// TIA Portal project "S7-1500 ile Giyotin Makası Kontrolü Uygulaması" (V18)

(* hardware
DEVICE "S7-1500/ET200MP station_1"  S7-1500 station
   slot 0: "Rail_0"  Rack  6ES7 590-1***0-0AA0
   slot 1: "PLC_1"  CPU 1512C-1 PN  6ES7 512-1CK01-0AB0  V2.8
      slot 3: "CPU display_1"  6ES7591-1AA00-0AA0
      slot 32768: "PROFINET interface_1"  X1
         slot 32769: "Port_1"  X1 P1
         slot 32770: "Port_2"  X1 P2
      slot 34817: "Virtual CP interface port_1"  Virtual CP interface port  Virtual CP interface port
DEVICE "HMI_1"  KTP700 Basic PN
   slot 0: "HMI_1"  KTP700 Basic PN  6AV2 123-2GB03-0AX0  14.0.1.0
   slot 1: "HMI_RT_1"  KTP700 Basic PN  6AV2 123-2GB03-0AX0  14.0.1.0
   slot 5: "HMI_1.IE_CP_1"  PROFINET Interface  14.0.1.0
      slot 1: "PROFINET Interface_1"  PROFINET Interface
         slot 1: "Port_1"  Port
*)

// ===== PLC "PLC_1"  CPU 1512C-1 PN =====

VAR_GLOBAL   // PLC tag table "Default tag table"
   "Stop" AT %M0.0 : Bool;
   "İleri" AT %Q0.0 : Bool;
   "Sınır Anahtarı" AT %M0.1 : Bool;
   "Start_1" AT %M0.2 : Bool;
   "Geri" AT %Q0.1 : Bool;
   "Start_2" AT %M0.3 : Bool;
END_VAR

ORGANIZATION_BLOCK "Main"   // OB1, LAD, ProgramCycle
TITLE = "Main Program Sweep (Cycle)"
{ S7_Optimized_Access := 'TRUE' }
VERSION : 0.1
   VAR_INPUT
      Initial_Call : Bool;   // Initial call of this OB
      Remanence : Bool;   // =True, if remanent data are available
   END_VAR
BEGIN

REGION Network 1: Giyotin makasın ileri-geri yön kontrolü yapılacaktır.
   // 2 starta basınca sistem giyorin sistemi çalışacaktır.
   // Stop+Sınır anahtarı aktif olunca sistem geri gidecek.
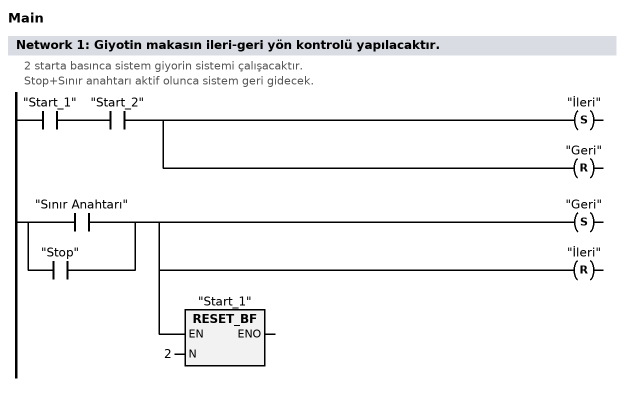
   // no SCL statement known for RBitfield: written as a call
   IF "Start_1" AND "Start_2" THEN
       "İleri" := TRUE;
       "Geri" := FALSE;
   END_IF;
   IF "Sınır Anahtarı" OR "Stop" THEN
       "Geri" := TRUE;
       "İleri" := FALSE;
       RESET_BF(operand := "Start_1", n := 2);
   END_IF;
END_REGION
END_ORGANIZATION_BLOCK

(* ===== HMI "HMI_RT_1" =====
system functions are stored by id; their names below are inferred from use
connection "Connection_1": ETHERNET, SMART_S7_1500_OMS
connection "HMI_Connection_1": ETHERNET, SMART_S7_1500_OMS

HMI tags "Default tag table"
   "Tag_ScreenNumber" : UInt, internal
   "Start_1" : Bool = PLC Start_1 AT %M0.2, 100 ms
   "Start_2" : Bool = PLC Start_2 AT %M0.3, 100 ms
   "Stop" : Bool = PLC Stop AT %M0.0, 100 ms
   "Sınır Anahtarı" : Bool = PLC "Sınır Anahtarı" AT %M0.1, 100 ms
   "İleri" : Bool = PLC İleri AT %Q0.0, 100 ms
   "Geri" : Bool = PLC Geri AT %Q0.1, 100 ms

graphic list "Geri Hareket": 0 'Graphic_22'; 1 'Graphic_23'

graphic list "İleri Hareket": 0 'Graphic_21'; 1 'Graphic_20'

Template "Template_1" 800x480
   Button "Exit" at 714,429 size 71x50; TextOff 'Exit'; PictureOff "ExitRuntime_KTP700_Basic_PN_TR"; PictureOn "ExitRuntime_KTP700_Basic_PN_TR"
      on Release: StopRuntime(0)
   Button "Language" at 614,429 size 71x50; TextOff 'Language'; PictureOff "ToggleLanguage_KTP700_Basic_PN_TR"; PictureOn "ToggleLanguage_KTP700_Basic_PN_TR"
      on Release: function_fb9197e8(-1)
   Button "Log on" at 514,429 size 71x50; TextOff 'Log on'; PictureOff "Login_KTP700_Basic_PN_TR"; PictureOn "Login_KTP700_Basic_PN_TR"
      on Release: function_a2a04561()
   Button "Alarms" at 114,429 size 71x50; TextOff 'Alarms'; PictureOff "AlarmDisplay_KTP700_Basic_PN_TR"; PictureOn "AlarmDisplay_KTP700_Basic_PN_TR"
      on Release: function_ef3f5d25("Alarm window_Unacknowledged", -1)
   Button "Start screen" at 14,429 size 71x50; TextOff 'Start screen'; PictureOff "NavigateHome_KTP700_Basic_PN_TR"; PictureOn "NavigateHome_KTP700_Basic_PN_TR"
      on Release: ActivateScreen("Root screen", 0)
   SymbolicIOField "Symbolic_IO_Field_Screen" at 93,9 size 600x33; TextOff '0'; TextOn '1'; TextList "TextList_ScreenNames"
      ProcessValue <- "Tag_ScreenNumber"
      on Change: ActivateScreenByNumber("Tag_ScreenNumber", 0)
   DateTimeField "HmiScreenItemData" at 695,25 size 105x25
   DateTimeField "HmiScreenItemData_1" at 695,0 size 105x25
   GraphicView "Logo" at 0,0 size 91x51; Picture "Logo of HMI_1"

screen "Root screen" 800x480, template "Template_1"
   on GenerateScreen: SetTag("Tag_ScreenNumber", 1)
   Button "Button_1" at 331,258 size 128x49; TextOff 'Start_2'
      on Click: InvertBit("Start_2")
   Button "Button_2" at 330,385 size 129x50; TextOff 'Sınır Anahtarı'
      on Press: SetBit("Sınır Anahtarı")
      on Release: ResetBit("Sınır Anahtarı")
   Button "Button_3" at 331,322 size 129x50; TextOff 'Stop'
      on Press: SetBit("Stop")
      on Release: ResetBit("Stop")
   Button "Button_4" at 330,193 size 129x50; TextOff 'Start_1'
      on Click: InvertBit("Start_1")
   GraphicIOField "Graphic I/O field_1" at 234,95 size 96x81; PictureList "Geri Hareket"
      ProcessValue <- "Geri"
      Visibility <- "Geri"
   GraphicIOField "Graphic I/O field_2" at 460,95 size 96x81; PictureList "İleri Hareket"
      ProcessValue <- "Tag_ScreenNumber"
      Visibility <- "İleri"
   GraphicView "Graphic view_1" at 343,93 size 109x83; Picture "Graphic_24"
*)